% RSLogix 500 project COIN.RSS, saved by version 8.10.00.18 %
PROJECT "COIN"    % processor: SLC 500, 1747-L531 %

PROGRAM FILES
  LAD 2   30 rungs

DATA FILES
  O0 OUTPUT  9 elements
  I1 INPUT  9 elements
  S2 STATUS  83 elements
  B3 BINARY  2 elements
  T4 TIMER  14 elements
  C5 COUNTER  1 elements
  R6 CONTROL  1 elements
  N7 INTEGER  1 elements
  F8 FLOAT  1 elements

LADDER 2
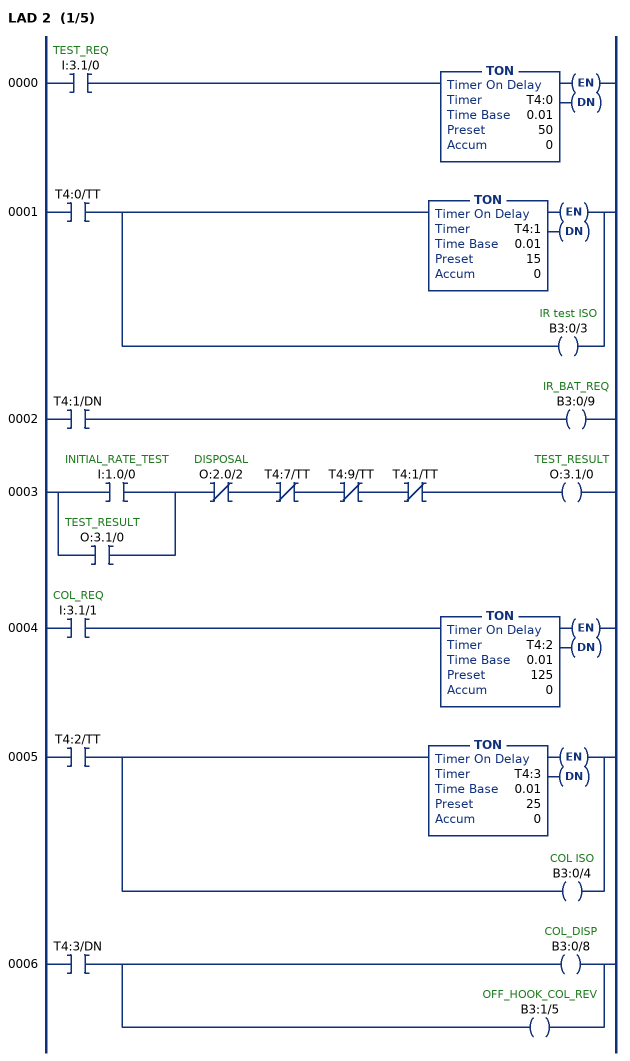
% Rung: 0 %
SOR XIC I:3.1/0 TON T4:0 0.01 50 0 EOR
%   I:3.1/0  TEST_REQ %
% Rung: 1 %
SOR XIC T4:0/TT BST TON T4:1 0.01 15 0 NXB OTE B3:0/3 BND EOR
%   B3:0/3  "IR test ISO" %
% Rung: 2 %
SOR XIC T4:1/DN OTE B3:0/9 EOR
%   B3:0/9  IR_BAT_REQ %
% Rung: 3 %
SOR BST XIC I:1.0/0 NXB XIC O:3.1/0 BND XIO O:2.0/2 XIO T4:7/TT XIO T4:9/TT XIO T4:1/TT OTE O:3.1/0 EOR
%   I:1.0/0  INITIAL_RATE_TEST %
%   O:3.1/0  TEST_RESULT %
%   O:2.0/2  DISPOSAL %
% Rung: 4 %
SOR XIC I:3.1/1 TON T4:2 0.01 125 0 EOR
%   I:3.1/1  COL_REQ %
% Rung: 5 %
SOR XIC T4:2/TT BST TON T4:3 0.01 25 0 NXB OTE B3:0/4 BND EOR
%   B3:0/4  "COL ISO" %
% Rung: 6 %
SOR XIC T4:3/DN BST OTE B3:0/8 NXB OTE B3:1/5 BND EOR
%   B3:0/8  COL_DISP %
%   B3:1/5  OFF_HOOK_COL_REV %

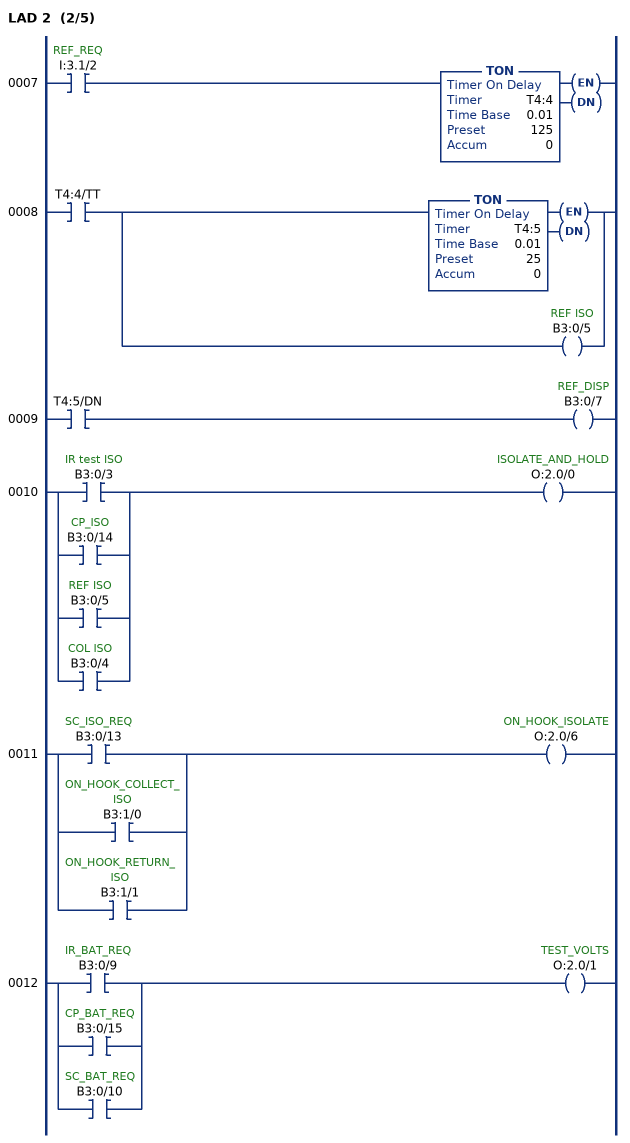
% Rung: 7 %
SOR XIC I:3.1/2 TON T4:4 0.01 125 0 EOR
%   I:3.1/2  REF_REQ %
% Rung: 8 %
SOR XIC T4:4/TT BST TON T4:5 0.01 25 0 NXB OTE B3:0/5 BND EOR
%   B3:0/5  "REF ISO" %
% Rung: 9 %
SOR XIC T4:5/DN OTE B3:0/7 EOR
%   B3:0/7  REF_DISP %
% Rung: 10 %
SOR BST XIC B3:0/3 NXB XIC B3:0/14 NXB XIC B3:0/5 NXB XIC B3:0/4 BND OTE O:2.0/0 EOR
%   B3:0/3  "IR test ISO" %
%   B3:0/14  CP_ISO %
%   B3:0/5  "REF ISO" %
%   B3:0/4  "COL ISO" %
%   O:2.0/0  ISOLATE_AND_HOLD %
% Rung: 11 %
SOR BST XIC B3:0/13 NXB XIC B3:1/0 NXB XIC B3:1/1 BND OTE O:2.0/6 EOR
%   B3:0/13  SC_ISO_REQ %
%   B3:1/0  ON_HOOK_COLLECT_ISO %
%   B3:1/1  ON_HOOK_RETURN_ISO %
%   O:2.0/6  ON_HOOK_ISOLATE %
% Rung: 12 %
SOR BST XIC B3:0/9 NXB XIC B3:0/15 NXB XIC B3:0/10 BND OTE O:2.0/1 EOR
%   B3:0/9  IR_BAT_REQ %
%   B3:0/15  CP_BAT_REQ %
%   B3:0/10  SC_BAT_REQ %
%   O:2.0/1  TEST_VOLTS %

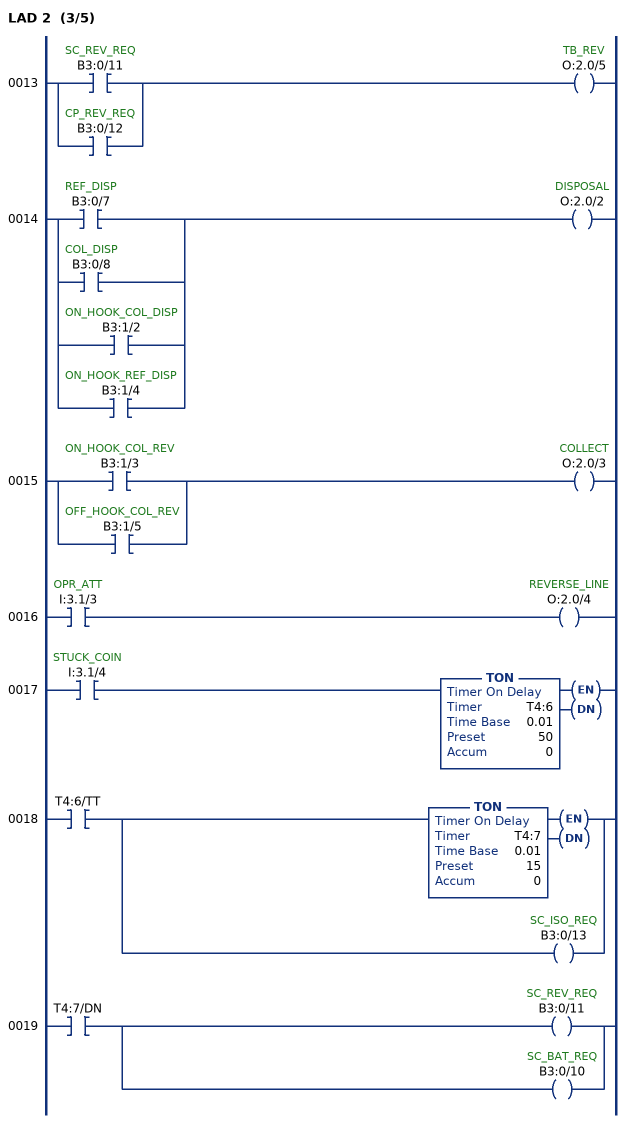
% Rung: 13 %
SOR BST XIC B3:0/11 NXB XIC B3:0/12 BND OTE O:2.0/5 EOR
%   B3:0/11  SC_REV_REQ %
%   B3:0/12  CP_REV_REQ %
%   O:2.0/5  TB_REV %
% Rung: 14 %
SOR BST XIC B3:0/7 NXB XIC B3:0/8 NXB XIC B3:1/2 NXB XIC B3:1/4 BND OTE O:2.0/2 EOR
%   B3:0/7  REF_DISP %
%   B3:0/8  COL_DISP %
%   B3:1/2  ON_HOOK_COL_DISP %
%   B3:1/4  ON_HOOK_REF_DISP %
%   O:2.0/2  DISPOSAL %
% Rung: 15 %
SOR BST XIC B3:1/3 NXB XIC B3:1/5 BND OTE O:2.0/3 EOR
%   B3:1/3  ON_HOOK_COL_REV %
%   B3:1/5  OFF_HOOK_COL_REV %
%   O:2.0/3  COLLECT %
% Rung: 16 %
SOR XIC I:3.1/3 OTE O:2.0/4 EOR
%   I:3.1/3  OPR_ATT %
%   O:2.0/4  REVERSE_LINE %
% Rung: 17 %
SOR XIC I:3.1/4 TON T4:6 0.01 50 0 EOR
%   I:3.1/4  STUCK_COIN %
% Rung: 18 %
SOR XIC T4:6/TT BST TON T4:7 0.01 15 0 NXB OTE B3:0/13 BND EOR
%   B3:0/13  SC_ISO_REQ %
% Rung: 19 %
SOR XIC T4:7/DN BST OTE B3:0/11 NXB OTE B3:0/10 BND EOR
%   B3:0/11  SC_REV_REQ %
%   B3:0/10  SC_BAT_REQ %

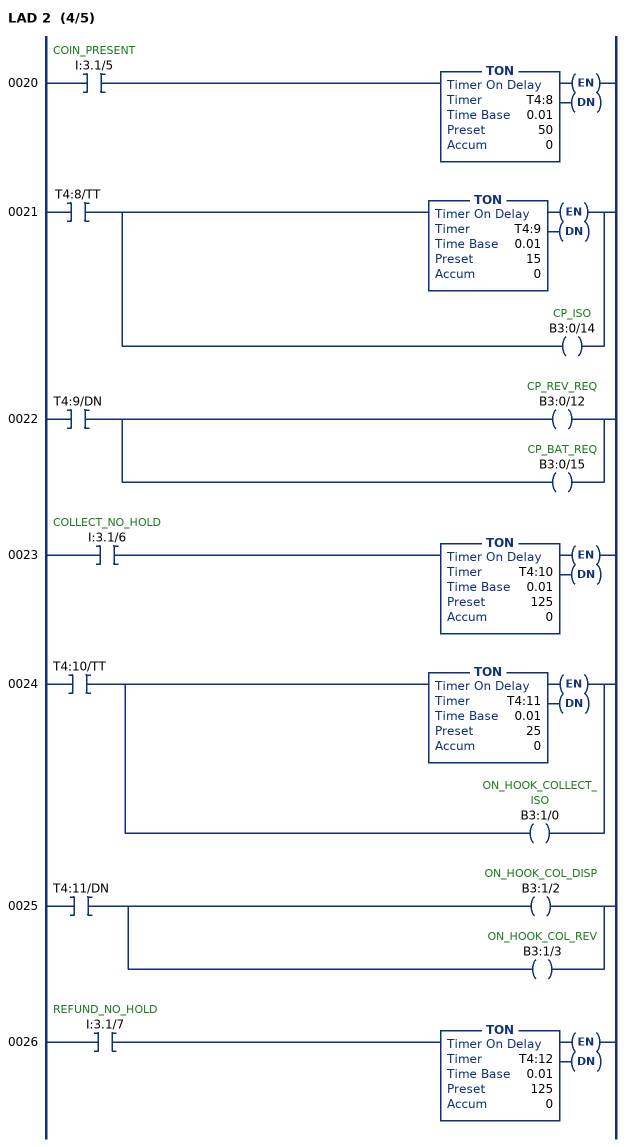
% Rung: 20 %
SOR XIC I:3.1/5 TON T4:8 0.01 50 0 EOR
%   I:3.1/5  COIN_PRESENT %
% Rung: 21 %
SOR XIC T4:8/TT BST TON T4:9 0.01 15 0 NXB OTE B3:0/14 BND EOR
%   B3:0/14  CP_ISO %
% Rung: 22 %
SOR XIC T4:9/DN BST OTE B3:0/12 NXB OTE B3:0/15 BND EOR
%   B3:0/12  CP_REV_REQ %
%   B3:0/15  CP_BAT_REQ %
% Rung: 23 %
SOR XIC I:3.1/6 TON T4:10 0.01 125 0 EOR
%   I:3.1/6  COLLECT_NO_HOLD %
% Rung: 24 %
SOR XIC T4:10/TT BST TON T4:11 0.01 25 0 NXB OTE B3:1/0 BND EOR
%   B3:1/0  ON_HOOK_COLLECT_ISO %
% Rung: 25 %
SOR XIC T4:11/DN BST OTE B3:1/2 NXB OTE B3:1/3 BND EOR
%   B3:1/2  ON_HOOK_COL_DISP %
%   B3:1/3  ON_HOOK_COL_REV %
% Rung: 26 %
SOR XIC I:3.1/7 TON T4:12 0.01 125 0 EOR
%   I:3.1/7  REFUND_NO_HOLD %

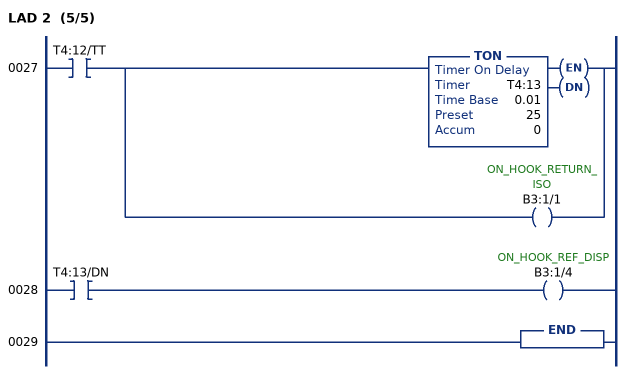
% Rung: 27 %
SOR XIC T4:12/TT BST TON T4:13 0.01 25 0 NXB OTE B3:1/1 BND EOR
%   B3:1/1  ON_HOOK_RETURN_ISO %
% Rung: 28 %
SOR XIC T4:13/DN OTE B3:1/4 EOR
%   B3:1/4  ON_HOOK_REF_DISP %
% Rung: 29 %
SOR END EOR

DATA TABLE (non-zero values as saved)
DATA T4
% .PRE .ACC %
% T4:0 % 50 0
% T4:1 % 15 0
% T4:2 % 125 0
% T4:3 % 25 0
% T4:4 % 125 0
% T4:5 % 25 0
% T4:6 % 50 0
% T4:7 % 15 0
% T4:8 % 50 0
% T4:9 % 15 0
% T4:10 % 125 0
% T4:11 % 25 0
% T4:12 % 125 0
% T4:13 % 25 0
